FUNCTION F_Log : bool
VAR_INPUT
	str1		:STRING;
END_VAR
VAR
	rTrig:R_TRIG;
	
END_VAR



rTrig(CLK:= TRUE, Q=> );

IF (rTrig.Q) THEN 
	GVL_General.LogBufferIndex := GVL_General.LogBufferIndex + 1;

	str1 := CONCAT(STR1:= ':',STR2:= str1);
	str1 := CONCAT(STR1:= F_TimeNow(), STR2:= str1);
	str1 := CONCAT(STR1:= str1,STR2 := '$n');

	GVL_General.LogBufferArray[GVL_General.LogBufferIndex] := str1;
	rTrig(CLK:= FALSE, Q=> );
END_IF

(*GVL_General.LogBufferIndex := GVL_General.LogBufferIndex + 1;

str1 := CONCAT(STR1:= ':',STR2:= str1);
str1 := CONCAT(STR1:= F_TimeNow(), STR2:= str1);
str1 := CONCAT(STR1:= str1,STR2 := '$n');

GVL_General.LogBufferArray[GVL_General.LogBufferIndex] := str1;  *)

END_FUNCTION

(* stored: Version 1.1.0.1, ProductVersion 3.1.4022.16
   POU F_Log: Id {9a415fdc-fd5a-4695-bb1f-7978a429ab50}, SpecialFunc None *)
